TYPE union_State :
UNION
	uiState		: UINT;
	eState		: enum_State;
END_UNION
END_TYPE

(* stored: Version 1.1.0.1
   DUT union_State: Id {118e705c-c32c-4c6a-8887-686c353c4081} *)
